TYPE T_Ctrl_SIf_HPS_Par :
STRUCT
	/// Timeout communication at Datachannel
	udiTimeOutRead_ms: UDINT;
	/// [ms] Time to wait for starting a new drive
	udiTimeDriveStart_ms: UDINT;
	/// [ms] Time to wait for stopping a new drive
	udiTimeDriveStop_ms: UDINT;
	/// [ms] Interval buffer filling
	udiIntervalBufferFilling_ms: UDINT;
END_STRUCT
END_TYPE

(* stored: Version 1.1.0.1, ProductVersion 3.1.0.19
   DUT T_Ctrl_SIf_HPS_Par: Id {0c82fbbf-ad8a-44fb-aa73-aaeab4b43a22} *)
